(*

short summary
=================
Test implementation of IAlarm interface for unit testing.
Simulates alarm behavior with throw, acknowledge, and pending state tracking.

.. <legal notes>

legal notes
=================
| SPDX-FileCopyrightText: © 2025 ekvip automation GmbH <info@ekvip.de>
| SPDX-License-Identifier: Apache-2.0
| For details check: Apache-2.0_

.. _Apache-2.0: https://www.apache.org/licenses/LICENSE-2.0

.. </legal notes>

methods and properties
=========================

*)
FUNCTION_BLOCK TestAlarm EXTENDS CNM_AbstractObject.Object IMPLEMENTS CNM_MessageInterfaces.IAlarm
VAR
	wasThrownMarker : BOOL;
	isPendingValue : BOOL;
	acknowledgeCounter : INT;
END_VAR

(*

short summary
=================
Acknowledges the alarm and clears the pending state.
Increments the acknowledge counter for test verification.

.. <legal notes>

legal notes
=================
| SPDX-FileCopyrightText: © 2025 ekvip automation GmbH <info@ekvip.de>
| SPDX-License-Identifier: Apache-2.0
| For details check: Apache-2.0_

.. _Apache-2.0: https://www.apache.org/licenses/LICENSE-2.0

.. </legal notes>

*)
METHOD acknowledge : CNM_ReturnTypes.SingleExecutionResult
THIS^.isPendingValue := FALSE;
THIS^.acknowledgeCounter := THIS^.acknowledgeCounter + 1;
acknowledge := CNM_ReturnTypes.SingleExecutionResult.SUCCESS;
END_METHOD

PROPERTY className : CNM_AbstractObject.ClassName
GET
className := 'TestAlarm';
END_GET
END_PROPERTY

(*

short summary
=================
This method clears the message and resets it to a predefined state.

.. <legal notes>

legal notes
=================
| SPDX-FileCopyrightText: © 2024 ekvip automation GmbH <info@ekvip.de>
| SPDX-License-Identifier: Apache-2.0
| For details check: Apache-2.0_

.. _Apache-2.0: https://www.apache.org/licenses/LICENSE-2.0

.. </legal notes>

*)
METHOD clear
END_METHOD


(*

short summary
=================
This property returns the dto of the message containing the data.

.. <legal notes>

legal notes
=================
| SPDX-FileCopyrightText: © 2024 ekvip automation GmbH <info@ekvip.de>
| SPDX-License-Identifier: Apache-2.0
| For details check: Apache-2.0_

.. _Apache-2.0: https://www.apache.org/licenses/LICENSE-2.0

.. </legal notes>

*)
PROPERTY dto : CNM_MessageInterfaces.IMessageDto
GET
END_GET
END_PROPERTY

(*

short summary
=================
Invokes the action associated with this interface.

.. <legal notes>

legal notes
=================
| SPDX-FileCopyrightText: © 2024 ekvip automation GmbH <info@ekvip.de>
| SPDX-License-Identifier: Apache-2.0
| For details check: Apache-2.0_

.. _Apache-2.0: https://www.apache.org/licenses/LICENSE-2.0

.. </legal notes>

parameters
=================

*)
METHOD invoke : CNM_CommandInterfaces.CNM_ReturnTypes.SingleExecutionResult
END_METHOD

PROPERTY isPending : BOOL
GET
isPending := THIS^.isPendingValue;
END_GET
END_PROPERTY

(*

short summary
=================
Resets all alarm state variables to initial values.

.. <legal notes>

legal notes
=================
| SPDX-FileCopyrightText: © 2025 ekvip automation GmbH <info@ekvip.de>
| SPDX-License-Identifier: Apache-2.0
| For details check: Apache-2.0_

.. _Apache-2.0: https://www.apache.org/licenses/LICENSE-2.0

.. </legal notes>

*)
METHOD reset
THIS^.wasThrownMarker := FALSE;
THIS^.isPendingValue := FALSE;
THIS^.acknowledgeCounter := 0;
END_METHOD

(*

short summary
=================
Throws the test alarm by setting pending state.
Tracks that the alarm was thrown for test verification.

.. <legal notes>

legal notes
=================
| SPDX-FileCopyrightText: © 2025 ekvip automation GmbH <info@ekvip.de>
| SPDX-License-Identifier: Apache-2.0
| For details check: Apache-2.0_

.. _Apache-2.0: https://www.apache.org/licenses/LICENSE-2.0

.. </legal notes>

*)
METHOD throw
THIS^.wasThrownMarker := TRUE;
THIS^.isPendingValue := TRUE;
END_METHOD

PROPERTY wasThrown : BOOL
GET
wasThrown := THIS^.wasThrownMarker;
END_GET
SET
THIS^.wasThrownMarker := wasThrown;
END_SET
END_PROPERTY

END_FUNCTION_BLOCK

(* stored: Version 1.1.0.1
   POU TestAlarm: Id {d0789012-789a-bcde-5678-901234562232}, SpecialFunc None
   Method acknowledge: Id {f2901234-9abc-ef01-789a-123456784454}
   Property className: Id {36345678-def0-3456-bcde-567890128898}
   Get Get: Id {47456789-ef01-4567-cdef-678901239909}
   Method clear: Id {b7665660-0c82-49fe-93a7-30a98be87b80}
   Property dto: Id {3f3eee17-d43c-4deb-a52c-b8ba931782e2}
   Get Get: Id {ec4290d5-2f10-48eb-b012-70d89442a7c9}
   Method invoke: Id {b322d326-6296-487b-93a5-a13e1dab9039}
   Property isPending: Id {14123456-bcde-1234-9abc-345678906676}
   Get Get: Id {25234567-cdef-2345-abcd-456789017787}
   Method reset: Id {03012345-abcd-0123-89ab-234567895565}
   Method throw: Id {e1890123-89ab-cdef-6789-012345673343}
   Property wasThrown: Id {db697f75-4673-4111-88bd-906d75162e92}
   Get Get: Id {7a1cff51-fc13-4d97-894d-1518b53cce43}
   Set Set: Id {d710f479-d61a-4106-8fa8-fbc77d5c44c4} *)
